{attribute 'OPC.UA.DA' := '1'}
{attribute 'OPC.UA.DA.StructuredType' := '1'}
TYPE WavelengthMsg :
STRUCT
	Id : EPowerIlluminationFlow;
	Wavelength : INT;
END_STRUCT
END_TYPE

(* stored: Version 1.1.0.1, ProductVersion 3.1.4024.3
   DUT WavelengthMsg: Id {28d1166c-5d67-4148-a0b1-7bdb0072c750} *)
